FUNCTION_BLOCK FB_Button
VAR_INPUT
END_VAR
VAR_OUTPUT
END_VAR
VAR
	bValue:					Bool;
END_VAR

PROPERTY PUBLIC P_Value : Bool
GET
P_Value:= bValue;
END_GET
END_PROPERTY

END_FUNCTION_BLOCK

(* stored: Version 1.1.0.1, ProductVersion 3.1.4024.12
   POU FB_Button: Id {f0bf445d-e7e9-047f-292f-1913811cf770}, SpecialFunc None
   Property P_Value: Id {791bd1dd-c417-0c32-3c36-c0924969df13}
   Get Get: Id {581e9463-ac2f-0620-058a-89326f94b997} *)
